FUNCTION_BLOCK FB_LampUpDown IMPLEMENTS I_Subject
VAR
	nLightLevel			:	USINT;
	_ipObserver			:	I_Observer;	
END_VAR

METHOD Attach
VAR_INPUT
	ipObserver		: I_Observer;
END_VAR
IF (ipObserver = 0) THEN
	RETURN;
END_IF
_ipObserver := ipObserver;
END_METHOD

METHOD Detach
_ipObserver := 0;
END_METHOD

// Reduces the control value by 1 in the range of 10 to 100. 
METHOD PUBLIC OneStepDown
nLightLevel := nLightLevel - 1;
IF (nLightLevel < 10) THEN
	nLightLevel := 10;
END_IF
IF (_ipObserver <> 0) THEN
	_ipObserver.Update(nLightLevel);
END_IF
END_METHOD

// Increments the control value by 1 in the range of 10 to 100.
METHOD PUBLIC OneStepUp
nLightLevel := nLightLevel + 1;
IF (nLightLevel > 100) THEN
	nLightLevel := 100;
END_IF
IF (_ipObserver <> 0) THEN
	_ipObserver.Update(nLightLevel);
END_IF
END_METHOD

// Toggles the control value between 0 and 100.
METHOD PUBLIC OnOff
IF (nLightLevel > 0) THEN
	nLightLevel := 0;
ELSE
	nLightLevel := 100;
END_IF
IF (_ipObserver <> 0) THEN
	_ipObserver.Update(nLightLevel);
end_IF
END_METHOD

END_FUNCTION_BLOCK

(* stored: Version 1.1.0.1, ProductVersion 3.1.4024.12
   POU FB_LampUpDown: Id {e5938590-1890-43a0-ba86-32547ab377e2}, SpecialFunc None
   Method Attach: Id {d670d29b-536a-4f65-a3ce-01855557f23a}
   Method Detach: Id {c4c4c396-be35-4305-a634-3561a50debfd}
   Method OneStepDown: Id {eccc8046-24a1-4940-82a7-bde5c3e6c0ab}
   Method OneStepUp: Id {bdc89d87-e6d0-409f-9392-70820315cfad}
   Method OnOff: Id {4e5634f0-9545-430f-86b8-452bc4855175} *)
